Omron CX-Programmer project NewProject (CX-Programmer 9.61)

# PLC KEEP: CP1L M
; TEST FUNGSI KEEP

## Global symbols (name address type ; comment)
0.00 BOOL  ; START
0.01 BOOL  ; RESET
100.00 BOOL  ; OUT

## Program NewProgram1 (cyclic task 0)

### Section Section1

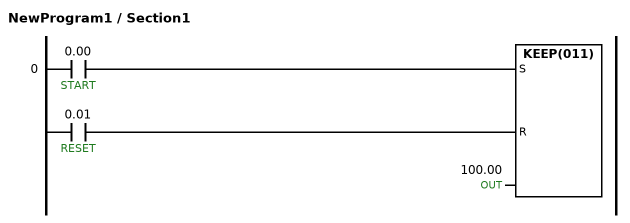
; rung 0
LD 0.00  ; START
LD 0.01  ; RESET
KEEP(011) 100.00  ; OUT

### Section END
; rung 0
END(001)